(* PLC project display_management, Dassault Systèmes ControlBuild 2024x *)
(* stored: creationDateTime 2023-10-03T11:13:48-01:00 *)

FUNCTION_BLOCK tni_clock.display_management
  VAR_INPUT
    hh : SINT := 0;
    mn : SINT := 0;
    sec : SINT := 0;
  END_VAR
  VAR_INPUT
    tick : BOOL := false;
  END_VAR
  VAR_INPUT
    pressure : INT := 0;
  END_VAR
  VAR_IN_OUT
    B1 : BOOL := false;
    B2 : BOOL := false;
    B3 : BOOL := false;
    B4 : BOOL := false;
  END_VAR
  VAR_OUTPUT
    displayValue : ARRAY[1..8] OF BYTE := [8(0)];
  END_VAR
  VAR_OUTPUT
    switchOnLight : BOOL := false;
  END_VAR
  VAR
    displayTime : REAL := 0.0;
    lampSwitchOnTime : REAL := 0.0;
  END_VAR
  VAR CONSTANT
    pulseTime : DINT := 10;
  END_VAR

(***** time/pressure selection button push management ******)
(* button push temporisation for 10s *)
IF ((B3 OR displayTime > 0.0) AND tick) THEN
(* one RE of tick every 2 cycles. CLOCK_PERIOD corresponds to quartz frequency *)
	displayTime := displayTime + (CLOCK_PERIOD/1000000.0 * 2.0); 
END_IF;
IF (displayTime > 10.0) OR NOT B3 THEN
	B3 := FALSE;
	displayTime := 0.0;
END_IF;


IF B3 THEN
(***** Pressure display *****)
(* Every digit take the ascii value corresponding to the measure *)
	displayValue[1] := 48 + pressure/1000;
	displayValue[2] := 48 + (pressure - ((pressure/1000)*1000))/100;
	displayValue[3] := 48 + (pressure - ((pressure/1000)*1000) - (((pressure - ((pressure/1000)*1000))/100)*100))/10;
	displayValue[4] := 48 + (pressure - ((pressure/1000)*1000) - (((pressure - ((pressure/1000)*1000))/100)*100) - (((pressure - ((pressure/1000)*1000) - (((pressure - ((pressure/1000)*1000))/100)*100))/10)*10));
	displayValue[5] := 32 (* space *);
	displayValue[6] := 104 (* $h *);
	displayValue[7] := 80 (* $P *);
	displayValue[8] := 97 (* $a *);

ELSE
(***** Time display *****)
(* Every digit take the ascii value corresponding to the current time*)
	displayValue[1] := 48 + hh/10;
	displayValue[2] := 48 + (hh - ((hh/10)*10));
	displayValue[3] := 58 (* $: *);
	displayValue[4] := 48 + mn/10;
	displayValue[5] := 48 + (mn - ((mn/10)*10));
	displayValue[6] := 58 (* $: *);
	displayValue[7] := 48 + sec/10;
	displayValue[8] := 48 + (sec - ((sec/10)*10));
END_IF;

(**** Lighting management ****)
(* button push temporisation for 3s *)
IF ((B4 OR lampSwitchOnTime >0) AND tick) THEN
(* one RE of tick every 2 cycles. CLOCK_PERIOD corresponds to quartz frequency *)
	lampSwitchOnTime := lampSwitchOnTime + (CLOCK_PERIOD/1000000 * 2.0); 
END_IF;
IF (lampSwitchOnTime > 3) THEN
	B4 := FALSE;
	lampSwitchOnTime:= 0;
END_IF;
switchOnLight := lampSwitchOnTime>0.0;
END_FUNCTION_BLOCK
